// TIA Portal V20 export
DATA_BLOCK "DB_SystemSimu"   // DB30
// stored: Access Published, MemoryReserve 100, Namespace Global
   VAR
      TriggerSensor : Struct
         Line : Struct
            ProductionLine : Struct
               Conveyor : Array[_.gminProductionLine.._.gmaxProductionLine] of Bool;
            END_STRUCT;
            EmptyLine : Struct
               Conveyor : Array[_.gminEmptyLine.._.gmaxEmptyLine] of Bool;
            END_STRUCT;
            PackedLine : Struct
               Conveyor : Array[_.gminPackedLine.._.gmaxPackedLine] of Bool;
            END_STRUCT;
         END_STRUCT;
      END_STRUCT;
      TriggerFault : Struct
         Line : Struct
            ProductionLine : Struct
               Conveyor : Array[_.gminProductionLine.._.gmaxProductionLine] of Bool;
            END_STRUCT;
            EmptyLine : Struct
               Conveyor : Array[_.gminEmptyLine.._.gmaxEmptyLine] of Bool;
            END_STRUCT;
            PackedLine : Struct
               Conveyor : Array[_.gminPackedLine.._.gmaxPackedLine] of Bool;
            END_STRUCT;
         END_STRUCT;
      END_STRUCT;
      Fire : Bool;
      DatamanResultsAvailable : Bool;
   END_VAR
BEGIN
   // TriggerSensor.Line.ProductionLine.Conveyor[1001] : AS1.1.1
   // TriggerSensor.Line.ProductionLine.Conveyor[1002] : AS1.1.2
   // TriggerFault.Line.ProductionLine.Conveyor[1001] : AS1.1.1
   // TriggerFault.Line.ProductionLine.Conveyor[1002] : AS1.1.2
END_DATA_BLOCK
